Fanuc KAREL source: kt00531.KL

-- PROVISIONAL review KL for V1013-1; original PC SHA256 3ded10278548ee09b23769f82d52e4dacc976b7d5e6c517b65f7f04960379f09
-- Incomplete behavior may be omitted. Consult companion uncertainty JSON. Do not deploy.
PROGRAM KT00531
%NOLOCKGROUP
-- UNRESOLVED_DECL P1 type=000106
-- UNRESOLVED_DECL P2 type=000199
-- UNRESOLVED_DECL OUT type=000106
BEGIN
  -- UNRESOLVED_PC offsets 5-20; opcodes 2E,22,32,35
  -- UNRESOLVED_PC offsets 25-64; opcodes 49,7E,49,7E,60,7E,4A
  -- UNRESOLVED_PC offsets 69-73; opcodes 7F
END KT00531
